FUNCTION_BLOCK WOOD_DECODER
  {SET_ATTRIBUTE(OpcUa, SERVICE)}
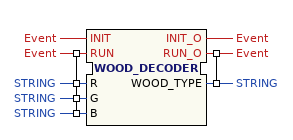
  EVENT_INPUT
    INIT;
    RUN WITH R, G, B; {SET_ATTRIBUTE(OpcUa, Method)}
  END_EVENT
  EVENT_OUTPUT
    INIT_O;
    RUN_O WITH WOOD_TYPE;
  END_EVENT
  VAR_INPUT
    R : STRING;
    G : STRING;
    B : STRING;
  END_VAR
  VAR_OUTPUT
    WOOD_TYPE : STRING;
  END_VAR
END_FUNCTION_BLOCK
